# EPICS autosave request: support/ebrick/2-2-3/iocBoot/iocebrick/autosave/auto_positions.req
## eBrick positions
file ebrick_positions.req P=$(P)
